FUNCTION_BLOCK FB_Workplate EXTENDS FB_SlotTarget
VAR_INPUT
END_VAR
VAR_OUTPUT
END_VAR
VAR
	rCollHeight			: REAL;
	bCalcCollHeight		: BOOL;
	iter				: FB_ObjCollectIteratorDeep;
	pTarget				: POINTER TO FB_TargetBase;
	stAbsPosCenter		: ST_3DPoint;
	fbRectangle			: FB_Rectangle;
	nParentSlotNr		: UINT;		//Workplate befindet sich zwar an keinem Slot, aber virtuell in der GUI (am Root)
END_VAR

IF bCalcCollHeight THEN
	bCalcCollHeight := FALSE;
	fbRectangle(X1:=0.0, Y1:=0.0, X2:=stDimension.Width, Y2:=stDimension.Depth);
	pTarget := M_GetHighestTarget(fbRectAngle,0.0);
	IF pTarget > 0 THEN
		IF pTarget^.P_rAbsFreeHeight > P_rAbsFreeHeight THEN
			rCollHeight := pTarget^.P_rAbsFreeHeight + 1000.0;
		ELSE
			rCollHeight := P_rAbsFreeHeight + 1000.0;
		END_IF
	ELSE
		rCollHeight := P_rAbsFreeHeight + 1000.0;
	END_IF
END_IF

METHOD FB_init : BOOL
VAR_INPUT
	bInitRetains : BOOL; // if TRUE, the retain variables are initialized (warm start / cold start)
	bInCopyCode : BOOL;  // if TRUE, the instance afterwards gets moved into the copy code (online change)
END_VAR
eObjectType := E_ObjectType.OBJECTTYPE_Workplate;
eObjectGroup := E_ObjectGroup.OBJECTGROUP_Target;
END_METHOD

METHOD M_AddChild : ERRORID
VAR_INPUT
	pObject : POINTER TO FB_Object;
	nSlotNr	: UINT;
	nIndex 	: INT;
END_VAR
//Kann alle Targets aufnehmen
IF pObject > 0 THEN
	IF pObject^.M_bIsGroup(E_ObjectGroup.OBJECTGROUP_Target) THEN
		M_AddChild := SUPER^.M_AddChild(pObject,nSlotNr,nIndex);
	ELSE
		M_AddChild := E_ErrorIdObjMgmt.ERRORID_InvalidParentObject;
	END_IF
ELSE
	M_AddChild := E_ErrorIdObjMgmt.ERRORID_InvalidParentObject;
END_IF
END_METHOD

METHOD M_ClearAllProps
VAR_INPUT
	bIgnoreParent : BOOL; //Es wird das gesamte OD gelöscht. -> Zeiger auf Parent nicht mehr gültig!
END_VAR
SUPER^.M_ClearAllProps(bIgnoreParent);
rCollHeight := 0;
END_METHOD

METHOD M_GetAllProps : ERRORID
VAR_INPUT
	refCmdData : REFERENCE TO  ST_CmdData;
END_VAR
SUPER^.M_GetAllProps(refCmdData);

refCmdData.n32Data[1] := nParentSlotNr;
END_METHOD

METHOD M_SetAllProps : ERRORID
VAR_INPUT
	refCmdData : REFERENCE TO  ST_CmdData;
END_VAR
M_SetAllProps := SUPER^.M_SetAllProps(refCmdData);
IF M_SetAllProps > 0 THEN
	RETURN;
END_IF

nParentSlotNr := DINT_TO_UINT(refCmdData.n32Data[1]);
END_METHOD

PROPERTY P_bCalcCollisHeight : BOOL
SET
bCalcCollHeight := P_bCalcCollisHeight;
END_SET
END_PROPERTY

PROPERTY P_nParentSlotNr : UINT
GET
P_nParentSlotNr := nParentSlotNr;
END_GET
END_PROPERTY

PROPERTY P_rCollHeight : REAL
GET
P_rCollHeight := rCollHeight;
END_GET
SET
rCollHeight := P_rCollHeight;
END_SET
END_PROPERTY

END_FUNCTION_BLOCK

(* stored: Version 1.1.0.1, ProductVersion 3.1.4022.18
   POU FB_Workplate: Id {5f9e774b-fbeb-4995-af82-5e1c4a7d3ee5}, SpecialFunc None
   Method FB_init: Id {4647c8d4-1292-4106-a7ef-22cd432239e1}
   Method M_AddChild: Id {0c363073-83ab-4c55-b772-9e45e35f773d}
   Method M_ClearAllProps: Id {29e69567-d46b-4d41-afc8-0ab8ddbf98db}
   Method M_GetAllProps: Id {d59b6009-164c-4995-b4ae-ddf127d5601a}
   Method M_SetAllProps: Id {26c005d3-d78c-4d2b-aba3-7ba86939f4b1}
   Property P_bCalcCollisHeight: Id {19baa40b-2a28-4e28-a903-c6b8eea972b9}
   Set Set: Id {c69c5f60-f7ea-4eeb-abee-f118c10ce474}
   Property P_nParentSlotNr: Id {5df26b9f-f086-4a45-9a77-f46a438b4b62}
   Get Get: Id {a8373210-5c56-4652-97b7-5ee889a47b0f}
   Property P_rCollHeight: Id {48f2e55f-e824-44ea-9881-1c197cd65386}
   Get Get: Id {ea52a64a-f421-4ff9-a8a5-b84eb602ccf4}
   Set Set: Id {c4274f4d-2da8-47dd-87de-6d26508ff102} *)
